{attribute 'GeneratedUsingTerminal: EL6001-0000-0020'}
{attribute addProperty BoxType "EL6001-0000-0020"}
{attribute addProperty Id "StatusAT %I*Status_3D84275F8Data_InAT %I*ARRAY[0..49] OF UINT100"}
{attribute addProperty CRC "1924718055"}
{attribute addProperty Size "108"}
TYPE COM_ext_inputs_1F197B20 :
STRUCT
	{attribute addProperty Name "Status"}
	Status AT %I* : Status_3D84275F;
	{attribute addProperty Name "Data_In"}
	Data_In AT %I* : ARRAY[0..49] OF UINT;
END_STRUCT
END_TYPE

(* stored: Version 1.2.0.0, ProductVersion 3.1.4024.9
   DUT COM_ext_inputs_1F197B20: Id {124ba976-63f8-4153-962f-77fd277e02eb} *)
